	MoveL Offs(p0,47.0,21.0, 0), v10, z5, tool0;
	MoveL Offs(p0,47.0,18.0, 0), v10, z5, tool0;
	MoveL Offs(p0,46.0,18.0, 0), v10, z5, tool0;
	MoveL Offs(p0,44.0,18.0, 0), v10, z5, tool0;
	MoveL Offs(p0,43.0,18.0, 0), v10, z5, tool0;
	MoveL Offs(p0,43.0,19.0, 0), v10, z5, tool0;
	MoveL Offs(p0,43.0,19.0, 0), v10, z5, tool0;
	MoveL Offs(p0,42.0,19.0, 0), v10, z5, tool0;
	MoveL Offs(p0,39.0,19.0, 0), v10, z5, tool0;
	MoveL Offs(p0,37.0,20.0, 0), v10, z5, tool0;
	MoveL Offs(p0,37.0,20.0, 0), v10, z5, tool0;
	MoveL Offs(p0,36.0,21.0, 0), v10, z5, tool0;
	MoveL Offs(p0,36.0,22.0, 0), v10, z5, tool0;
	MoveL Offs(p0,36.0,22.0, 0), v10, z5, tool0;
	MoveL Offs(p0,37.0,23.0, 0), v10, z5, tool0;
	MoveL Offs(p0,38.0,24.0, 0), v10, z5, tool0;
	MoveL Offs(p0,40.0,25.0, 0), v10, z5, tool0;
	MoveL Offs(p0,42.0,26.0, 0), v10, z5, tool0;
	MoveL Offs(p0,42.0,26.0, 0), v10, z5, tool0;
	MoveL Offs(p0,43.0,26.0, 0), v10, z5, tool0;
	MoveL Offs(p0,43.0,26.0, 0), v10, z5, tool0;
	MoveL Offs(p0,44.0,26.0, 0), v10, z5, tool0;
	MoveL Offs(p0,44.0,26.0, 0), v10, z5, tool0;
	MoveL Offs(p0,46.0,27.0, 0), v10, z5, tool0;
	MoveL Offs(p0,47.0,27.0, 0), v10, z5, tool0;
	MoveL Offs(p0,47.0,27.0, 0), v10, z5, tool0;
	MoveL Offs(p0,47.0,27.0, 0), v10, z5, tool0;
	MoveL Offs(p0,47.0,27.0, 0), v10, z5, tool0;
	MoveL Offs(p0,47.0,27.0, 0), v10, z5, tool0;
	MoveL Offs(p0,47.0,27.0, 0), v10, z5, tool0;
	MoveJ Offs(p0,47.0,27.0, 20), v10, z1, tool0;
	MoveJ Offs(p0,31.0,25.0, 20), v10, z1, tool0;
	MoveJ Offs(p0,31.0,25.0, 0), v10, z1, tool0;
	MoveL Offs(p0,32.0,24.0, 0), v10, z5, tool0;
	MoveL Offs(p0,32.0,22.0, 0), v10, z5, tool0;
	MoveL Offs(p0,31.0,20.0, 0), v10, z5, tool0;
	MoveL Offs(p0,31.0,20.0, 0), v10, z5, tool0;
	MoveL Offs(p0,31.0,19.0, 0), v10, z5, tool0;
	MoveL Offs(p0,31.0,19.0, 0), v10, z5, tool0;
	MoveL Offs(p0,29.0,19.0, 0), v10, z5, tool0;
	MoveL Offs(p0,28.0,19.0, 0), v10, z5, tool0;
	MoveL Offs(p0,26.0,21.0, 0), v10, z5, tool0;
	MoveL Offs(p0,25.0,22.0, 0), v10, z5, tool0;
	MoveL Offs(p0,25.0,23.0, 0), v10, z5, tool0;
	MoveL Offs(p0,24.0,23.0, 0), v10, z5, tool0;
	MoveL Offs(p0,24.0,24.0, 0), v10, z5, tool0;
	MoveL Offs(p0,24.0,24.0, 0), v10, z5, tool0;
	MoveL Offs(p0,24.0,25.0, 0), v10, z5, tool0;
	MoveL Offs(p0,24.0,25.0, 0), v10, z5, tool0;
	MoveL Offs(p0,27.0,26.0, 0), v10, z5, tool0;
	MoveL Offs(p0,28.0,25.0, 0), v10, z5, tool0;
	MoveL Offs(p0,29.0,25.0, 0), v10, z5, tool0;
	MoveL Offs(p0,29.0,25.0, 0), v10, z5, tool0;
	MoveL Offs(p0,30.0,25.0, 0), v10, z5, tool0;
	MoveL Offs(p0,31.0,25.0, 0), v10, z5, tool0;
	MoveL Offs(p0,31.0,25.0, 0), v10, z5, tool0;
	MoveJ Offs(p0,31.0,25.0, 20), v10, z1, tool0;
	MoveJ Offs(p0,74.0,16.0, 20), v10, z1, tool0;
	MoveJ Offs(p0,74.0,16.0, 0), v10, z1, tool0;
	MoveL Offs(p0,76.0,15.0, 0), v10, z5, tool0;
	MoveL Offs(p0,78.0,15.0, 0), v10, z5, tool0;
	MoveL Offs(p0,79.0,15.0, 0), v10, z5, tool0;
	MoveL Offs(p0,80.0,15.0, 0), v10, z5, tool0;
	MoveL Offs(p0,81.0,14.0, 0), v10, z5, tool0;
	MoveL Offs(p0,83.0,14.0, 0), v10, z5, tool0;
	MoveL Offs(p0,84.0,14.0, 0), v10, z5, tool0;
	MoveL Offs(p0,85.0,15.0, 0), v10, z5, tool0;
	MoveL Offs(p0,86.0,15.0, 0), v10, z5, tool0;
	MoveL Offs(p0,88.0,15.0, 0), v10, z5, tool0;
	MoveL Offs(p0,89.0,15.0, 0), v10, z5, tool0;
	MoveL Offs(p0,89.0,15.0, 0), v10, z5, tool0;
	MoveL Offs(p0,89.0,15.0, 0), v10, z5, tool0;
	MoveL Offs(p0,89.0,15.0, 0), v10, z5, tool0;
	MoveL Offs(p0,88.0,13.0, 0), v10, z5, tool0;
	MoveL Offs(p0,87.0,12.0, 0), v10, z5, tool0;
	MoveL Offs(p0,86.0,11.0, 0), v10, z5, tool0;
	MoveL Offs(p0,86.0,10.0, 0), v10, z5, tool0;
	MoveL Offs(p0,85.0,10.0, 0), v10, z5, tool0;
	MoveL Offs(p0,84.0,9.0, 0), v10, z5, tool0;
	MoveL Offs(p0,83.0,8.0, 0), v10, z5, tool0;
	MoveL Offs(p0,81.0,7.0, 0), v10, z5, tool0;
	MoveL Offs(p0,78.0,5.0, 0), v10, z5, tool0;
	MoveL Offs(p0,75.0,4.0, 0), v10, z5, tool0;
	MoveL Offs(p0,72.0,3.0, 0), v10, z5, tool0;
	MoveL Offs(p0,69.0,3.0, 0), v10, z5, tool0;
	MoveL Offs(p0,67.0,2.0, 0), v10, z5, tool0;
	MoveL Offs(p0,64.0,3.0, 0), v10, z5, tool0;
	MoveL Offs(p0,62.0,3.0, 0), v10, z5, tool0;
	MoveL Offs(p0,59.0,4.0, 0), v10, z5, tool0;
	MoveL Offs(p0,57.0,5.0, 0), v10, z5, tool0;
	MoveL Offs(p0,55.0,6.0, 0), v10, z5, tool0;
	MoveL Offs(p0,54.0,7.0, 0), v10, z5, tool0;
	MoveL Offs(p0,54.0,8.0, 0), v10, z5, tool0;
	MoveL Offs(p0,53.0,8.0, 0), v10, z5, tool0;
	MoveL Offs(p0,53.0,9.0, 0), v10, z5, tool0;
	MoveL Offs(p0,53.0,9.0, 0), v10, z5, tool0;
	MoveL Offs(p0,52.0,9.0, 0), v10, z5, tool0;
	MoveL Offs(p0,52.0,10.0, 0), v10, z5, tool0;
	MoveL Offs(p0,53.0,12.0, 0), v10, z5, tool0;
	MoveL Offs(p0,54.0,13.0, 0), v10, z5, tool0;
	MoveL Offs(p0,56.0,14.0, 0), v10, z5, tool0;
	MoveL Offs(p0,58.0,15.0, 0), v10, z5, tool0;
	MoveL Offs(p0,59.0,15.0, 0), v10, z5, tool0;
	MoveL Offs(p0,61.0,16.0, 0), v10, z5, tool0;
	MoveL Offs(p0,64.0,17.0, 0), v10, z5, tool0;
	MoveL Offs(p0,66.0,17.0, 0), v10, z5, tool0;
	MoveL Offs(p0,68.0,17.0, 0), v10, z5, tool0;
	MoveL Offs(p0,71.0,17.0, 0), v10, z5, tool0;
	MoveL Offs(p0,71.0,17.0, 0), v10, z5, tool0;
	MoveL Offs(p0,72.0,17.0, 0), v10, z5, tool0;
	MoveL Offs(p0,72.0,16.0, 0), v10, z5, tool0;
	MoveL Offs(p0,73.0,16.0, 0), v10, z5, tool0;
	MoveL Offs(p0,74.0,16.0, 0), v10, z5, tool0;
	MoveL Offs(p0,74.0,16.0, 0), v10, z5, tool0;
	MoveJ Offs(p0,74.0,16.0, 20), v10, z1, tool0;
	MoveJ Offs(p0,27.0,13.0, 20), v10, z1, tool0;
	MoveJ Offs(p0,27.0,13.0, 0), v10, z1, tool0;
	MoveL Offs(p0,29.0,11.0, 0), v10, z5, tool0;
	MoveL Offs(p0,30.0,11.0, 0), v10, z5, tool0;
	MoveL Offs(p0,30.0,11.0, 0), v10, z5, tool0;
	MoveL Offs(p0,31.0,10.0, 0), v10, z5, tool0;
	MoveL Offs(p0,32.0,10.0, 0), v10, z5, tool0;
	MoveL Offs(p0,32.0,9.0, 0), v10, z5, tool0;
	MoveL Offs(p0,33.0,8.0, 0), v10, z5, tool0;
	MoveL Offs(p0,33.0,8.0, 0), v10, z5, tool0;
	MoveL Offs(p0,35.0,5.0, 0), v10, z5, tool0;
	MoveL Offs(p0,34.0,5.0, 0), v10, z5, tool0;
	MoveL Offs(p0,31.0,6.0, 0), v10, z5, tool0;
	MoveL Offs(p0,30.0,7.0, 0), v10, z5, tool0;
	MoveL Offs(p0,29.0,8.0, 0), v10, z5, tool0;
	MoveL Offs(p0,27.0,8.0, 0), v10, z5, tool0;
	MoveL Offs(p0,26.0,9.0, 0), v10, z5, tool0;
	MoveL Offs(p0,25.0,10.0, 0), v10, z5, tool0;
	MoveL Offs(p0,24.0,10.0, 0), v10, z5, tool0;
	MoveL Offs(p0,24.0,11.0, 0), v10, z5, tool0;
	MoveL Offs(p0,22.0,13.0, 0), v10, z5, tool0;
	MoveL Offs(p0,25.0,13.0, 0), v10, z5, tool0;
	MoveL Offs(p0,25.0,13.0, 0), v10, z5, tool0;
	MoveL Offs(p0,26.0,13.0, 0), v10, z5, tool0;
	MoveL Offs(p0,26.0,13.0, 0), v10, z5, tool0;
	MoveL Offs(p0,27.0,13.0, 0), v10, z5, tool0;
	MoveL Offs(p0,27.0,13.0, 0), v10, z5, tool0;
	MoveJ Offs(p0,27.0,13.0, 20), v10, z1, tool0;
	MoveJ Offs(p0,49.0,10.0, 20), v10, z1, tool0;
	MoveJ Offs(p0,49.0,10.0, 0), v10, z1, tool0;
	MoveL Offs(p0,51.0,8.0, 0), v10, z5, tool0;
	MoveL Offs(p0,52.0,8.0, 0), v10, z5, tool0;
	MoveL Offs(p0,52.0,8.0, 0), v10, z5, tool0;
	MoveL Offs(p0,53.0,7.0, 0), v10, z5, tool0;
	MoveL Offs(p0,55.0,5.0, 0), v10, z5, tool0;
	MoveL Offs(p0,55.0,5.0, 0), v10, z5, tool0;
	MoveL Offs(p0,56.0,4.0, 0), v10, z5, tool0;
	MoveL Offs(p0,56.0,4.0, 0), v10, z5, tool0;
	MoveL Offs(p0,56.0,4.0, 0), v10, z5, tool0;
	MoveL Offs(p0,55.0,2.0, 0), v10, z5, tool0;
	MoveL Offs(p0,54.0,1.0, 0), v10, z5, tool0;
	MoveL Offs(p0,52.0,1.0, 0), v10, z5, tool0;
	MoveL Offs(p0,51.0,1.0, 0), v10, z5, tool0;
	MoveL Offs(p0,49.0,1.0, 0), v10, z5, tool0;
	MoveL Offs(p0,48.0,1.0, 0), v10, z5, tool0;
	MoveL Offs(p0,46.0,1.0, 0), v10, z5, tool0;
	MoveL Offs(p0,45.0,2.0, 0), v10, z5, tool0;
	MoveL Offs(p0,43.0,2.0, 0), v10, z5, tool0;
	MoveL Offs(p0,41.0,3.0, 0), v10, z5, tool0;
	MoveL Offs(p0,40.0,3.0, 0), v10, z5, tool0;
	MoveL Offs(p0,39.0,4.0, 0), v10, z5, tool0;
	MoveL Offs(p0,38.0,4.0, 0), v10, z5, tool0;
	MoveL Offs(p0,38.0,5.0, 0), v10, z5, tool0;
	MoveL Offs(p0,37.0,5.0, 0), v10, z5, tool0;
	MoveL Offs(p0,36.0,6.0, 0), v10, z5, tool0;
	MoveL Offs(p0,36.0,6.0, 0), v10, z5, tool0;
	MoveL Offs(p0,35.0,7.0, 0), v10, z5, tool0;
	MoveL Offs(p0,34.0,8.0, 0), v10, z5, tool0;
	MoveL Offs(p0,35.0,9.0, 0), v10, z5, tool0;
	MoveL Offs(p0,38.0,10.0, 0), v10, z5, tool0;
	MoveL Offs(p0,39.0,10.0, 0), v10, z5, tool0;
	MoveL Offs(p0,40.0,10.0, 0), v10, z5, tool0;
	MoveL Offs(p0,41.0,10.0, 0), v10, z5, tool0;
	MoveL Offs(p0,41.0,10.0, 0), v10, z5, tool0;
	MoveL Offs(p0,43.0,10.0, 0), v10, z5, tool0;
	MoveL Offs(p0,44.0,10.0, 0), v10, z5, tool0;
	MoveL Offs(p0,46.0,10.0, 0), v10, z5, tool0;
	MoveL Offs(p0,46.0,10.0, 0), v10, z5, tool0;
	MoveL Offs(p0,47.0,10.0, 0), v10, z5, tool0;
	MoveL Offs(p0,48.0,10.0, 0), v10, z5, tool0;
	MoveL Offs(p0,48.0,10.0, 0), v10, z5, tool0;
	MoveL Offs(p0,48.0,10.0, 0), v10, z5, tool0;
	MoveL Offs(p0,49.0,10.0, 0), v10, z5, tool0;
	MoveL Offs(p0,49.0,10.0, 0), v10, z5, tool0;
	MoveL Offs(p0,49.0,10.0, 0), v10, z5, tool0;
	MoveJ Offs(p0,49.0,10.0, 20), v10, z1, tool0;
	MoveJ Offs(p0,119.0,121.0, 20), v10, z1, tool0;
	MoveJ Offs(p0,119.0,121.0, 0), v10, z1, tool0;
	MoveL Offs(p0,119.0,119.0, 0), v10, z5, tool0;
	MoveL Offs(p0,119.0,118.0, 0), v10, z5, tool0;
	MoveL Offs(p0,119.0,118.0, 0), v10, z5, tool0;
	MoveL Offs(p0,119.0,118.0, 0), v10, z5, tool0;
	MoveL Offs(p0,120.0,119.0, 0), v10, z5, tool0;
	MoveL Offs(p0,120.0,120.0, 0), v10, z5, tool0;
	MoveL Offs(p0,120.0,121.0, 0), v10, z5, tool0;
	MoveL Offs(p0,120.0,121.0, 0), v10, z5, tool0;
	MoveL Offs(p0,119.0,122.0, 0), v10, z5, tool0;
	MoveL Offs(p0,119.0,122.0, 0), v10, z5, tool0;
	MoveL Offs(p0,119.0,122.0, 0), v10, z5, tool0;
	MoveL Offs(p0,119.0,121.0, 0), v10, z5, tool0;
	MoveJ Offs(p0,119.0,121.0, 20), v10, z1, tool0;
	MoveJ Offs(p0,119.0,109.0, 20), v10, z1, tool0;
	MoveJ Offs(p0,119.0,109.0, 0), v10, z1, tool0;
	MoveL Offs(p0,116.0,107.0, 0), v10, z5, tool0;
	MoveL Offs(p0,116.0,107.0, 0), v10, z5, tool0;
	MoveL Offs(p0,116.0,106.0, 0), v10, z5, tool0;
	MoveL Offs(p0,113.0,104.0, 0), v10, z5, tool0;
	MoveL Offs(p0,112.0,103.0, 0), v10, z5, tool0;
	MoveL Offs(p0,111.0,102.0, 0), v10, z5, tool0;
	MoveL Offs(p0,110.0,102.0, 0), v10, z5, tool0;
	MoveL Offs(p0,109.0,101.0, 0), v10, z5, tool0;
	MoveL Offs(p0,107.0,100.0, 0), v10, z5, tool0;
	MoveL Offs(p0,106.0,100.0, 0), v10, z5, tool0;
	MoveL Offs(p0,105.0,99.0, 0), v10, z5, tool0;
	MoveL Offs(p0,103.0,99.0, 0), v10, z5, tool0;
	MoveL Offs(p0,103.0,98.0, 0), v10, z5, tool0;
	MoveL Offs(p0,102.0,98.0, 0), v10, z5, tool0;
	MoveL Offs(p0,102.0,98.0, 0), v10, z5, tool0;
	MoveL Offs(p0,101.0,98.0, 0), v10, z5, tool0;
	MoveL Offs(p0,101.0,98.0, 0), v10, z5, tool0;
	MoveL Offs(p0,99.0,97.0, 0), v10, z5, tool0;
	MoveL Offs(p0,98.0,97.0, 0), v10, z5, tool0;
	MoveL Offs(p0,98.0,97.0, 0), v10, z5, tool0;
	MoveL Offs(p0,98.0,96.0, 0), v10, z5, tool0;
	MoveL Offs(p0,97.0,96.0, 0), v10, z5, tool0;
	MoveL Offs(p0,97.0,96.0, 0), v10, z5, tool0;
	MoveL Offs(p0,97.0,95.0, 0), v10, z5, tool0;
	MoveL Offs(p0,99.0,92.0, 0), v10, z5, tool0;
	MoveL Offs(p0,99.0,91.0, 0), v10, z5, tool0;
	MoveL Offs(p0,100.0,90.0, 0), v10, z5, tool0;
	MoveL Offs(p0,101.0,88.0, 0), v10, z5, tool0;
	MoveL Offs(p0,103.0,87.0, 0), v10, z5, tool0;
	MoveL Offs(p0,104.0,85.0, 0), v10, z5, tool0;
	MoveL Offs(p0,106.0,82.0, 0), v10, z5, tool0;
	MoveL Offs(p0,108.0,80.0, 0), v10, z5, tool0;
	MoveL Offs(p0,109.0,78.0, 0), v10, z5, tool0;
	MoveL Offs(p0,110.0,77.0, 0), v10, z5, tool0;
	MoveL Offs(p0,111.0,75.0, 0), v10, z5, tool0;
	MoveL Offs(p0,112.0,74.0, 0), v10, z5, tool0;
	MoveL Offs(p0,113.0,72.0, 0), v10, z5, tool0;
	MoveL Offs(p0,114.0,70.0, 0), v10, z5, tool0;
	MoveL Offs(p0,115.0,68.0, 0), v10, z5, tool0;
	MoveL Offs(p0,116.0,66.0, 0), v10, z5, tool0;
	MoveL Offs(p0,117.0,62.0, 0), v10, z5, tool0;
	MoveL Offs(p0,118.0,61.0, 0), v10, z5, tool0;
	MoveL Offs(p0,119.0,60.0, 0), v10, z5, tool0;
	MoveL Offs(p0,120.0,58.0, 0), v10, z5, tool0;
	MoveL Offs(p0,120.0,57.0, 0), v10, z5, tool0;
	MoveL Offs(p0,121.0,56.0, 0), v10, z5, tool0;
	MoveL Offs(p0,121.0,56.0, 0), v10, z5, tool0;
	MoveL Offs(p0,122.0,55.0, 0), v10, z5, tool0;
	MoveL Offs(p0,122.0,55.0, 0), v10, z5, tool0;
	MoveL Offs(p0,124.0,54.0, 0), v10, z5, tool0;
	MoveL Offs(p0,125.0,54.0, 0), v10, z5, tool0;
	MoveL Offs(p0,127.0,54.0, 0), v10, z5, tool0;
	MoveL Offs(p0,128.0,55.0, 0), v10, z5, tool0;
	MoveL Offs(p0,130.0,56.0, 0), v10, z5, tool0;
	MoveL Offs(p0,132.0,57.0, 0), v10, z5, tool0;
	MoveL Offs(p0,134.0,58.0, 0), v10, z5, tool0;
	MoveL Offs(p0,136.0,59.0, 0), v10, z5, tool0;
	MoveL Offs(p0,138.0,60.0, 0), v10, z5, tool0;
	MoveL Offs(p0,140.0,61.0, 0), v10, z5, tool0;
	MoveL Offs(p0,141.0,62.0, 0), v10, z5, tool0;
	MoveL Offs(p0,143.0,64.0, 0), v10, z5, tool0;
	MoveL Offs(p0,144.0,64.0, 0), v10, z5, tool0;
	MoveL Offs(p0,145.0,65.0, 0), v10, z5, tool0;
	MoveL Offs(p0,145.0,65.0, 0), v10, z5, tool0;
	MoveL Offs(p0,145.0,66.0, 0), v10, z5, tool0;
	MoveL Offs(p0,145.0,66.0, 0), v10, z5, tool0;
	MoveL Offs(p0,145.0,67.0, 0), v10, z5, tool0;
	MoveL Offs(p0,145.0,68.0, 0), v10, z5, tool0;
	MoveL Offs(p0,145.0,69.0, 0), v10, z5, tool0;
	MoveL Offs(p0,144.0,72.0, 0), v10, z5, tool0;
	MoveL Offs(p0,143.0,74.0, 0), v10, z5, tool0;
	MoveL Offs(p0,142.0,76.0, 0), v10, z5, tool0;
	MoveL Offs(p0,140.0,78.0, 0), v10, z5, tool0;
	MoveL Offs(p0,139.0,81.0, 0), v10, z5, tool0;
	MoveL Offs(p0,137.0,84.0, 0), v10, z5, tool0;
	MoveL Offs(p0,136.0,87.0, 0), v10, z5, tool0;
	MoveL Offs(p0,134.0,89.0, 0), v10, z5, tool0;
	MoveL Offs(p0,132.0,92.0, 0), v10, z5, tool0;
	MoveL Offs(p0,130.0,96.0, 0), v10, z5, tool0;
	MoveL Offs(p0,129.0,98.0, 0), v10, z5, tool0;
	MoveL Offs(p0,127.0,101.0, 0), v10, z5, tool0;
	MoveL Offs(p0,126.0,103.0, 0), v10, z5, tool0;
	MoveL Offs(p0,125.0,105.0, 0), v10, z5, tool0;
	MoveL Offs(p0,124.0,106.0, 0), v10, z5, tool0;
	MoveL Offs(p0,123.0,107.0, 0), v10, z5, tool0;
	MoveL Offs(p0,122.0,108.0, 0), v10, z5, tool0;
	MoveL Offs(p0,122.0,108.0, 0), v10, z5, tool0;
	MoveL Offs(p0,121.0,109.0, 0), v10, z5, tool0;
	MoveL Offs(p0,119.0,109.0, 0), v10, z5, tool0;
	MoveL Offs(p0,119.0,109.0, 0), v10, z5, tool0;
	MoveL Offs(p0,119.0,109.0, 0), v10, z5, tool0;
	MoveL Offs(p0,119.0,109.0, 0), v10, z5, tool0;
	MoveJ Offs(p0,119.0,109.0, 20), v10, z1, tool0;
	MoveJ Offs(p0,121.0,108.0, 20), v10, z1, tool0;
	MoveJ Offs(p0,121.0,108.0, 0), v10, z1, tool0;
	MoveL Offs(p0,123.0,105.0, 0), v10, z5, tool0;
	MoveL Offs(p0,123.0,105.0, 0), v10, z5, tool0;
	MoveL Offs(p0,123.0,104.0, 0), v10, z5, tool0;
	MoveL Offs(p0,123.0,103.0, 0), v10, z5, tool0;
	MoveL Offs(p0,123.0,102.0, 0), v10, z5, tool0;
	MoveL Offs(p0,123.0,100.0, 0), v10, z5, tool0;
	MoveL Offs(p0,122.0,100.0, 0), v10, z5, tool0;
	MoveL Offs(p0,122.0,100.0, 0), v10, z5, tool0;
	MoveL Offs(p0,122.0,100.0, 0), v10, z5, tool0;
	MoveL Offs(p0,121.0,100.0, 0), v10, z5, tool0;
	MoveL Offs(p0,121.0,100.0, 0), v10, z5, tool0;
	MoveL Offs(p0,120.0,101.0, 0), v10, z5, tool0;
	MoveL Offs(p0,120.0,101.0, 0), v10, z5, tool0;
	MoveL Offs(p0,118.0,104.0, 0), v10, z5, tool0;
	MoveL Offs(p0,118.0,104.0, 0), v10, z5, tool0;
	MoveL Offs(p0,118.0,105.0, 0), v10, z5, tool0;
	MoveL Offs(p0,117.0,105.0, 0), v10, z5, tool0;
	MoveL Offs(p0,117.0,106.0, 0), v10, z5, tool0;
	MoveL Offs(p0,117.0,106.0, 0), v10, z5, tool0;
	MoveL Offs(p0,117.0,106.0, 0), v10, z5, tool0;
	MoveL Offs(p0,120.0,108.0, 0), v10, z5, tool0;
	MoveL Offs(p0,120.0,108.0, 0), v10, z5, tool0;
	MoveL Offs(p0,121.0,108.0, 0), v10, z5, tool0;
	MoveL Offs(p0,121.0,108.0, 0), v10, z5, tool0;
	MoveL Offs(p0,121.0,108.0, 0), v10, z5, tool0;
	MoveJ Offs(p0,121.0,108.0, 20), v10, z1, tool0;
	MoveJ Offs(p0,103.0,96.0, 20), v10, z1, tool0;
	MoveJ Offs(p0,103.0,96.0, 0), v10, z1, tool0;
	MoveL Offs(p0,104.0,94.0, 0), v10, z5, tool0;
	MoveL Offs(p0,104.0,93.0, 0), v10, z5, tool0;
	MoveL Offs(p0,105.0,93.0, 0), v10, z5, tool0;
	MoveL Offs(p0,105.0,92.0, 0), v10, z5, tool0;
	MoveL Offs(p0,105.0,91.0, 0), v10, z5, tool0;
	MoveL Offs(p0,105.0,91.0, 0), v10, z5, tool0;
	MoveL Offs(p0,105.0,90.0, 0), v10, z5, tool0;
	MoveL Offs(p0,102.0,90.0, 0), v10, z5, tool0;
	MoveL Offs(p0,102.0,91.0, 0), v10, z5, tool0;
	MoveL Offs(p0,101.0,91.0, 0), v10, z5, tool0;
	MoveL Offs(p0,100.0,92.0, 0), v10, z5, tool0;
	MoveL Offs(p0,100.0,93.0, 0), v10, z5, tool0;
	MoveL Offs(p0,99.0,95.0, 0), v10, z5, tool0;
	MoveL Offs(p0,99.0,95.0, 0), v10, z5, tool0;
	MoveL Offs(p0,99.0,96.0, 0), v10, z5, tool0;
	MoveL Offs(p0,99.0,96.0, 0), v10, z5, tool0;
	MoveL Offs(p0,99.0,96.0, 0), v10, z5, tool0;
	MoveL Offs(p0,100.0,97.0, 0), v10, z5, tool0;
	MoveL Offs(p0,102.0,97.0, 0), v10, z5, tool0;
	MoveL Offs(p0,102.0,97.0, 0), v10, z5, tool0;
	MoveL Offs(p0,102.0,97.0, 0), v10, z5, tool0;
	MoveL Offs(p0,103.0,96.0, 0), v10, z5, tool0;
	MoveL Offs(p0,103.0,96.0, 0), v10, z5, tool0;
	MoveJ Offs(p0,103.0,96.0, 20), v10, z1, tool0;
	MoveJ Offs(p0,131.0,90.0, 20), v10, z1, tool0;
	MoveJ Offs(p0,131.0,90.0, 0), v10, z1, tool0;
	MoveL Offs(p0,134.0,86.0, 0), v10, z5, tool0;
	MoveL Offs(p0,135.0,84.0, 0), v10, z5, tool0;
	MoveL Offs(p0,136.0,82.0, 0), v10, z5, tool0;
	MoveL Offs(p0,138.0,80.0, 0), v10, z5, tool0;
	MoveL Offs(p0,139.0,78.0, 0), v10, z5, tool0;
	MoveL Offs(p0,140.0,76.0, 0), v10, z5, tool0;
	MoveL Offs(p0,141.0,74.0, 0), v10, z5, tool0;
	MoveL Offs(p0,142.0,72.0, 0), v10, z5, tool0;
	MoveL Offs(p0,139.0,73.0, 0), v10, z5, tool0;
	MoveL Offs(p0,139.0,73.0, 0), v10, z5, tool0;
	MoveL Offs(p0,139.0,72.0, 0), v10, z5, tool0;
	MoveL Offs(p0,139.0,72.0, 0), v10, z5, tool0;
	MoveL Offs(p0,138.0,70.0, 0), v10, z5, tool0;
	MoveL Offs(p0,138.0,69.0, 0), v10, z5, tool0;
	MoveL Offs(p0,138.0,68.0, 0), v10, z5, tool0;
	MoveL Offs(p0,139.0,67.0, 0), v10, z5, tool0;
	MoveL Offs(p0,139.0,66.0, 0), v10, z5, tool0;
	MoveL Offs(p0,139.0,65.0, 0), v10, z5, tool0;
	MoveL Offs(p0,139.0,65.0, 0), v10, z5, tool0;
	MoveL Offs(p0,140.0,63.0, 0), v10, z5, tool0;
	MoveL Offs(p0,138.0,62.0, 0), v10, z5, tool0;
	MoveL Offs(p0,135.0,60.0, 0), v10, z5, tool0;
	MoveL Offs(p0,134.0,60.0, 0), v10, z5, tool0;
	MoveL Offs(p0,134.0,59.0, 0), v10, z5, tool0;
	MoveL Offs(p0,133.0,59.0, 0), v10, z5, tool0;
	MoveL Offs(p0,132.0,59.0, 0), v10, z5, tool0;
	MoveL Offs(p0,131.0,58.0, 0), v10, z5, tool0;
	MoveL Offs(p0,129.0,57.0, 0), v10, z5, tool0;
	MoveL Offs(p0,128.0,57.0, 0), v10, z5, tool0;
	MoveL Offs(p0,128.0,57.0, 0), v10, z5, tool0;
	MoveL Offs(p0,128.0,56.0, 0), v10, z5, tool0;
	MoveL Offs(p0,127.0,56.0, 0), v10, z5, tool0;
	MoveL Offs(p0,127.0,56.0, 0), v10, z5, tool0;
	MoveL Offs(p0,127.0,56.0, 0), v10, z5, tool0;
	MoveL Offs(p0,127.0,57.0, 0), v10, z5, tool0;
	MoveL Offs(p0,126.0,59.0, 0), v10, z5, tool0;
	MoveL Offs(p0,126.0,59.0, 0), v10, z5, tool0;
	MoveL Offs(p0,125.0,60.0, 0), v10, z5, tool0;
	MoveL Offs(p0,125.0,60.0, 0), v10, z5, tool0;
	MoveL Offs(p0,124.0,61.0, 0), v10, z5, tool0;
	MoveL Offs(p0,124.0,61.0, 0), v10, z5, tool0;
	MoveL Offs(p0,122.0,62.0, 0), v10, z5, tool0;
	MoveL Offs(p0,121.0,63.0, 0), v10, z5, tool0;
	MoveL Offs(p0,121.0,63.0, 0), v10, z5, tool0;
	MoveL Offs(p0,120.0,63.0, 0), v10, z5, tool0;
	MoveL Offs(p0,120.0,63.0, 0), v10, z5, tool0;
	MoveL Offs(p0,120.0,63.0, 0), v10, z5, tool0;
	MoveL Offs(p0,119.0,62.0, 0), v10, z5, tool0;
	MoveL Offs(p0,117.0,65.0, 0), v10, z5, tool0;
	MoveL Offs(p0,117.0,66.0, 0), v10, z5, tool0;
	MoveL Offs(p0,116.0,69.0, 0), v10, z5, tool0;
	MoveL Offs(p0,115.0,71.0, 0), v10, z5, tool0;
	MoveL Offs(p0,114.0,73.0, 0), v10, z5, tool0;
	MoveL Offs(p0,113.0,75.0, 0), v10, z5, tool0;
	MoveL Offs(p0,113.0,77.0, 0), v10, z5, tool0;
	MoveL Offs(p0,113.0,78.0, 0), v10, z5, tool0;
	MoveL Offs(p0,112.0,79.0, 0), v10, z5, tool0;
	MoveL Offs(p0,112.0,81.0, 0), v10, z5, tool0;
	MoveL Offs(p0,113.0,82.0, 0), v10, z5, tool0;
	MoveL Offs(p0,113.0,82.0, 0), v10, z5, tool0;
	MoveL Offs(p0,116.0,85.0, 0), v10, z5, tool0;
	MoveL Offs(p0,116.0,85.0, 0), v10, z5, tool0;
	MoveL Offs(p0,117.0,85.0, 0), v10, z5, tool0;
	MoveL Offs(p0,118.0,86.0, 0), v10, z5, tool0;
	MoveL Offs(p0,118.0,86.0, 0), v10, z5, tool0;
	MoveL Offs(p0,119.0,86.0, 0), v10, z5, tool0;
	MoveL Offs(p0,121.0,87.0, 0), v10, z5, tool0;
	MoveL Offs(p0,121.0,87.0, 0), v10, z5, tool0;
	MoveL Offs(p0,123.0,89.0, 0), v10, z5, tool0;
	MoveL Offs(p0,124.0,90.0, 0), v10, z5, tool0;
	MoveL Offs(p0,125.0,90.0, 0), v10, z5, tool0;
	MoveL Offs(p0,126.0,90.0, 0), v10, z5, tool0;
	MoveL Offs(p0,127.0,91.0, 0), v10, z5, tool0;
	MoveL Offs(p0,128.0,91.0, 0), v10, z5, tool0;
	MoveL Offs(p0,129.0,90.0, 0), v10, z5, tool0;
	MoveL Offs(p0,130.0,90.0, 0), v10, z5, tool0;
	MoveL Offs(p0,131.0,90.0, 0), v10, z5, tool0;
	MoveL Offs(p0,131.0,90.0, 0), v10, z5, tool0;
	MoveJ Offs(p0,131.0,90.0, 20), v10, z1, tool0;
	MoveJ Offs(p0,142.0,70.0, 20), v10, z1, tool0;
	MoveJ Offs(p0,142.0,70.0, 0), v10, z1, tool0;
	MoveL Offs(p0,144.0,68.0, 0), v10, z5, tool0;
	MoveL Offs(p0,144.0,68.0, 0), v10, z5, tool0;
	MoveL Offs(p0,144.0,67.0, 0), v10, z5, tool0;
	MoveL Offs(p0,143.0,65.0, 0), v10, z5, tool0;
	MoveL Offs(p0,143.0,65.0, 0), v10, z5, tool0;
	MoveL Offs(p0,142.0,65.0, 0), v10, z5, tool0;
	MoveL Offs(p0,142.0,65.0, 0), v10, z5, tool0;
	MoveL Offs(p0,142.0,65.0, 0), v10, z5, tool0;
	MoveL Offs(p0,140.0,66.0, 0), v10, z5, tool0;
	MoveL Offs(p0,139.0,67.0, 0), v10, z5, tool0;
	MoveL Offs(p0,139.0,68.0, 0), v10, z5, tool0;
	MoveL Offs(p0,139.0,70.0, 0), v10, z5, tool0;
	MoveL Offs(p0,139.0,71.0, 0), v10, z5, tool0;
	MoveL Offs(p0,139.0,71.0, 0), v10, z5, tool0;
	MoveL Offs(p0,140.0,71.0, 0), v10, z5, tool0;
	MoveL Offs(p0,140.0,72.0, 0), v10, z5, tool0;
	MoveL Offs(p0,140.0,71.0, 0), v10, z5, tool0;
	MoveL Offs(p0,141.0,71.0, 0), v10, z5, tool0;
	MoveL Offs(p0,141.0,71.0, 0), v10, z5, tool0;
	MoveL Offs(p0,142.0,70.0, 0), v10, z5, tool0;
	MoveL Offs(p0,142.0,70.0, 0), v10, z5, tool0;
	MoveJ Offs(p0,142.0,70.0, 20), v10, z1, tool0;
	MoveJ Offs(p0,122.0,61.0, 20), v10, z1, tool0;
	MoveJ Offs(p0,122.0,61.0, 0), v10, z1, tool0;
	MoveL Offs(p0,125.0,59.0, 0), v10, z5, tool0;
	MoveL Offs(p0,125.0,59.0, 0), v10, z5, tool0;
	MoveL Offs(p0,125.0,58.0, 0), v10, z5, tool0;
	MoveL Offs(p0,125.0,58.0, 0), v10, z5, tool0;
	MoveL Offs(p0,126.0,58.0, 0), v10, z5, tool0;
	MoveL Offs(p0,126.0,57.0, 0), v10, z5, tool0;
	MoveL Offs(p0,124.0,55.0, 0), v10, z5, tool0;
	MoveL Offs(p0,124.0,55.0, 0), v10, z5, tool0;
	MoveL Offs(p0,124.0,55.0, 0), v10, z5, tool0;
	MoveL Offs(p0,121.0,57.0, 0), v10, z5, tool0;
	MoveL Offs(p0,121.0,58.0, 0), v10, z5, tool0;
	MoveL Offs(p0,121.0,58.0, 0), v10, z5, tool0;
	MoveL Offs(p0,121.0,59.0, 0), v10, z5, tool0;
	MoveL Offs(p0,120.0,59.0, 0), v10, z5, tool0;
	MoveL Offs(p0,120.0,61.0, 0), v10, z5, tool0;
	MoveL Offs(p0,120.0,61.0, 0), v10, z5, tool0;
	MoveL Offs(p0,121.0,62.0, 0), v10, z5, tool0;
	MoveL Offs(p0,121.0,62.0, 0), v10, z5, tool0;
	MoveL Offs(p0,121.0,61.0, 0), v10, z5, tool0;
	MoveL Offs(p0,122.0,61.0, 0), v10, z5, tool0;
	MoveL Offs(p0,122.0,61.0, 0), v10, z5, tool0;
	MoveL Offs(p0,122.0,61.0, 0), v10, z5, tool0;
	MoveJ Offs(p0,122.0,61.0, 20), v10, z1, tool0;
	MoveJ Offs(p0,109.0,111.0, 20), v10, z1, tool0;
	MoveJ Offs(p0,109.0,111.0, 0), v10, z1, tool0;
	MoveL Offs(p0,108.0,109.0, 0), v10, z5, tool0;
	MoveL Offs(p0,108.0,109.0, 0), v10, z5, tool0;
	MoveL Offs(p0,109.0,111.0, 0), v10, z5, tool0;
	MoveJ Offs(p0,109.0,111.0, 20), v10, z1, tool0;
	MoveJ Offs(p0,99.0,106.0, 20), v10, z1, tool0;
	MoveJ Offs(p0,99.0,106.0, 0), v10, z1, tool0;
	MoveL Offs(p0,99.0,106.0, 0), v10, z5, tool0;
	MoveL Offs(p0,99.0,106.0, 0), v10, z5, tool0;
	MoveJ Offs(p0,99.0,106.0, 20), v10, z1, tool0;
	MoveJ Offs(p0,87.0,102.0, 20), v10, z1, tool0;
	MoveJ Offs(p0,87.0,102.0, 0), v10, z1, tool0;
	MoveL Offs(p0,89.0,101.0, 0), v10, z5, tool0;
	MoveL Offs(p0,90.0,101.0, 0), v10, z5, tool0;
	MoveL Offs(p0,90.0,101.0, 0), v10, z5, tool0;
	MoveL Offs(p0,90.0,101.0, 0), v10, z5, tool0;
	MoveL Offs(p0,92.0,101.0, 0), v10, z5, tool0;
	MoveL Offs(p0,91.0,101.0, 0), v10, z5, tool0;
	MoveL Offs(p0,88.0,102.0, 0), v10, z5, tool0;
	MoveL Offs(p0,88.0,103.0, 0), v10, z5, tool0;
	MoveL Offs(p0,88.0,103.0, 0), v10, z5, tool0;
	MoveL Offs(p0,87.0,102.0, 0), v10, z5, tool0;
	ENDPROC
ENDMODULE
